# EPICS substitutions: sdgEliteApp/Db/sdgElite-8.substitutions
file sdgElite01.template
{
pattern{ N, S }
       { 1, A }
       { 2, B }
       { 3, C }
       { 4, D }
       { 5, E }
       { 6, F }
       { 7, G }
       { 8, H }
}
